{attribute 'linkalways'} 
{attribute 'no_explicit_call' := 'This FB is a CLASS and must be accessed using methods or properties'}
{attribute 'enable_dynamic_creation'}
FUNCTION_BLOCK ABSTRACT Event IMPLEMENTS I_Event
VAR
	subscribers : SubscriberCollection;
END_VAR

METHOD PUBLIC AddSubscriber
VAR_INPUT
	Subscriber : I_Subscriber;
END_VAR
subscribers.Insert(Subscriber);
END_METHOD

METHOD PROTECTED NotifySubscribers
VAR
	count : UDINT;
	i : UDINT;
END_VAR
count := subscribers.Count;

IF count = 0 THEN
	RETURN;
END_IF

WHILE count > 0 DO 
	subscribers.GetByIndex(count - 1 ).Update(THIS^);
	count := count - 1;
END_WHILE
END_METHOD

METHOD PUBLIC RemoveSubscriber
VAR_INPUT
	Subscriber : I_Subscriber;
END_VAR
subscribers.Remove(Subscriber);
END_METHOD

END_FUNCTION_BLOCK

(* stored: Version 1.1.0.1, ProductVersion 3.1.4024.12
   POU Event: Id {ddead338-7e2e-0135-3c15-3a51bbfd1202}, SpecialFunc None
   Folder Protected: Id {68ff081f-c0b6-01c9-23b2-594f5b5c56dc}
   Method AddSubscriber: Id {4cf23379-b262-0e72-1b6b-d4b356376018}
   Method NotifySubscribers: Id {901b7e14-bced-0f65-2cc3-40c660cbdfa4}
   Method RemoveSubscriber: Id {aac87bfc-3f95-0ff1-34ce-4efce81a9d26} *)
